PROGRAM CaseStruct
VAR

END_VAR

CASE GVL.caseInput OF 
	0: // Initialisatie.
		GVL.ProductGedetecteerd1 := FALSE;	
		GVL.ProductGedetecteerd2 := FALSE;
		GVL.MotorStatus := FALSE;
		GVL.KlaarVoorVolgende := FALSE;
		IF GVL.ProductGedetecteerd1 AND NOT GVL.ProductGedetecteerd2 THEN
			GVL.caseInput := 1;
		END_IF
	1: // Product aan de start gedetecteerd.
		IF GVL.MotorStatus THEN
			GVL.caseInput := 2;
		END_IF
	2: // Product op het einde gedetecteerd.
		IF GVL.ProductGedetecteerd2 AND MAIN.Timer.ET > T#1S THEN
			GVL.caseInput := 3;
		END_IF
	3: // Programma weer afsluiten.
		IF MAIN.KlaarVoorVolgende THEN
			GVL.caseInput := 1;
			GVL.KlaarVoorVolgende := FALSE;
		END_IF
END_CASE

END_PROGRAM

(* stored: Version 1.1.0.1, ProductVersion 3.1.4024.12
   POU CaseStruct: Id {b01a3e46-c1c4-4cee-aff9-0d3865864dfe}, SpecialFunc None *)
